FUNCTION_BLOCK fbValvulaAbrirFecharPosicionar_Comunicacao (* Basic Function Block Type *)
  (* Standard: 61499-2 *)
  (* Version 0.0, 17/04/2026, Template *)
  PACKAGE Hidryco.HidrycoLib;
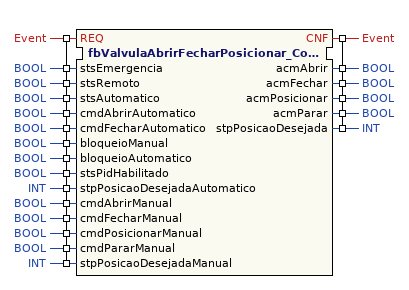
  EVENT_INPUT
    REQ WITH stsRemoto, stsAutomatico, cmdAbrirAutomatico, cmdFecharAutomatico, bloqueioManual, bloqueioAutomatico, stsPidHabilitado, stpPosicaoDesejadaAutomatico, cmdAbrirManual, cmdFecharManual, cmdPosicionarManual, stpPosicaoDesejadaManual, stsEmergencia, cmdPararManual; (* Normal Execution Request *)
  END_EVENT
  EVENT_OUTPUT
    CNF WITH acmAbrir, acmFechar, acmPosicionar, stpPosicaoDesejada, acmParar; (* Execution Confirmation *)
  END_EVENT
  VAR_INPUT
    stsEmergencia : BOOL;
    stsRemoto : BOOL;
    stsAutomatico : BOOL;
    cmdAbrirAutomatico : BOOL;
    cmdFecharAutomatico : BOOL;
    bloqueioManual : BOOL;
    bloqueioAutomatico : BOOL;
    stsPidHabilitado : BOOL;
    stpPosicaoDesejadaAutomatico : INT; (* Saida do PID *)
    cmdAbrirManual : BOOL;
    cmdFecharManual : BOOL;
    cmdPosicionarManual : BOOL;
    cmdPararManual : BOOL;
    stpPosicaoDesejadaManual : INT;
  END_VAR
  VAR_OUTPUT
    acmAbrir : BOOL;
    acmFechar : BOOL;
    acmPosicionar : BOOL;
    acmParar : BOOL;
    stpPosicaoDesejada : INT;
  END_VAR
  VAR
    prevStpAuto : INT;
  END_VAR
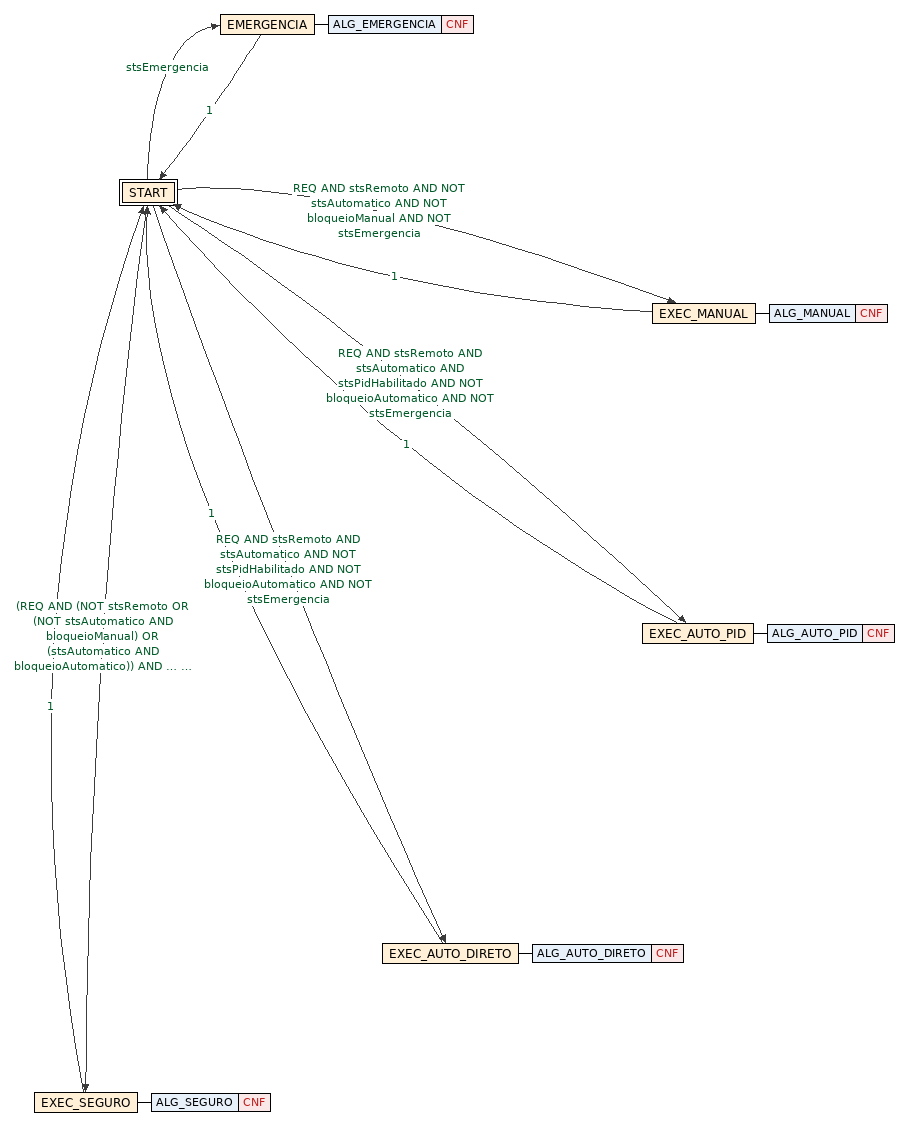
  EC_STATES
    START; (* Initial State *)
    EXEC_MANUAL : ALG_MANUAL -> CNF;
    EXEC_AUTO_PID : ALG_AUTO_PID -> CNF;
    EXEC_AUTO_DIRETO : ALG_AUTO_DIRETO -> CNF;
    EXEC_SEGURO : ALG_SEGURO -> CNF;
    EMERGENCIA : ALG_EMERGENCIA -> CNF;
  END_STATES
  EC_TRANSITIONS
    START TO EXEC_MANUAL := REQ AND stsRemoto AND NOT stsAutomatico AND NOT bloqueioManual AND NOT stsEmergencia;
    START TO EXEC_AUTO_PID := REQ AND stsRemoto AND stsAutomatico AND stsPidHabilitado AND NOT bloqueioAutomatico AND NOT stsEmergencia;
    START TO EXEC_AUTO_DIRETO := REQ AND stsRemoto AND stsAutomatico AND NOT stsPidHabilitado AND NOT bloqueioAutomatico AND NOT stsEmergencia;
    START TO EXEC_SEGURO := (REQ AND (NOT stsRemoto OR (NOT stsAutomatico AND bloqueioManual) OR (stsAutomatico AND bloqueioAutomatico)) AND NOT stsEmergencia);
    EXEC_MANUAL TO START := 1;
    EXEC_AUTO_PID TO START := 1;
    EXEC_AUTO_DIRETO TO START := 1;
    EXEC_SEGURO TO START := 1;
    START TO EMERGENCIA := stsEmergencia;
    EMERGENCIA TO START := 1;
  END_TRANSITIONS
  ALGORITHM ALG_MANUAL IN ST:
acmAbrir       := cmdAbrirManual;
acmFechar      := cmdFecharManual;
acmPosicionar  := cmdPosicionarManual;
acmParar		:= cmdPararManual;

IF cmdPosicionarManual THEN
    stpPosicaoDesejada := stpPosicaoDesejadaManual;
END_IF;
;
  END_ALGORITHM
  ALGORITHM ALG_AUTO_PID IN ST:
acmAbrir  := FALSE;
acmFechar := FALSE;
acmParar := FALSE;

IF stpPosicaoDesejadaAutomatico <> prevStpAuto THEN
    stpPosicaoDesejada := stpPosicaoDesejadaAutomatico;
    acmPosicionar      := TRUE;
ELSE
    acmPosicionar := FALSE;
END_IF;

prevStpAuto := stpPosicaoDesejadaAutomatico;
;
  END_ALGORITHM
  ALGORITHM ALG_AUTO_DIRETO IN ST:
acmAbrir       := cmdAbrirAutomatico;
acmFechar      := cmdFecharAutomatico;
acmPosicionar  := FALSE;
acmParar		:= FALSE;
;
  END_ALGORITHM
  ALGORITHM ALG_SEGURO IN ST:
acmAbrir       := FALSE;
acmFechar      := FALSE;
acmPosicionar  := FALSE;
acmParar		:= TRUE;
;
  END_ALGORITHM
  ALGORITHM ALG_EMERGENCIA IN ST:
acmAbrir       := FALSE;
acmFechar      := FALSE;
acmPosicionar  := FALSE;
acmParar		:= TRUE;

;
  END_ALGORITHM
END_FUNCTION_BLOCK
